(* CoDeSys 2.3 library: InfluxDB_1.0.0.0.lib *)
(* Libraries: BinaryTool_1.0.0.0.lib 25.8.19 15:16:50, TcpIp.lib 31.8.18 23:12:47, STANDARD.LIB 5.6.98 11:03:02, TcBase.lib 14.5.09 11:14:08, TcSystem.lib 7.6.16 10:01:22, TcUtilities.lib 3.2.16 15:08:58 *)

(* Global variable list: Global_Variables *)
VAR_GLOBAL
END_VAR
VAR_GLOBAL CONSTANT
	INFLUX_ROW_LEN : UINT := 350;
	INFLUX_FIFO_SIZE : UINT := 200;
	INFLUX_BUFFER_SIZE : UINT := 1200;
END_VAR

(* Data type *)
TYPE ST_InfluxDB_ConPar :
STRUCT
	sIpv4Address	: STRING	:= '127.0.0.1';
	uPort			: UINT		:= 8086;
	sHostName		: STRING	:= 'localhost';
	sDatabase		: STRING;
	sUser 			: STRING;
	sPassword		: STRING;
END_STRUCT
END_TYPE

(* Data type *)
TYPE ST_InfluxDB_Response :
STRUCT
	sContent		: T_MAXString;
	uCode		: UINT;
	bError		: BOOL;
END_STRUCT
END_TYPE

(* POU F_InfluxDb_BuildHttpPostRequest, ST *)
FUNCTION F_InfluxDb_BuildHttpPostRequest : BOOL
VAR_INPUT
	i_stInfluxDB_ConPar	: ST_InfluxDB_ConPar;
END_VAR
VAR_IN_OUT
	io_sInFluxData	: STRING(INFLUX_FIFO_SIZE);
	io_sBytesToSend	: FB_BinaryTool;
END_VAR
VAR
	nLength             : INT;
END_VAR
F_InfluxDb_BuildHttpPostRequest := F_BinaryTool_WriteString('POST ',io_sBytesToSend);
F_InfluxDb_BuildHttpPostRequest := F_InfluxDB_MakeURL(i_stInfluxDB_ConPar := i_stInfluxDB_ConPar, io_fbBinaryTool := io_sBytesToSend) AND F_InfluxDb_BuildHttpPostRequest;
F_InfluxDb_BuildHttpPostRequest := F_BinaryTool_WriteString(' HTTP/1.1$R$N',io_sBytesToSend) AND F_InfluxDb_BuildHttpPostRequest;
F_InfluxDb_BuildHttpPostRequest := F_BinaryTool_WriteString('Host: ',io_sBytesToSend) AND F_InfluxDb_BuildHttpPostRequest;
F_InfluxDb_BuildHttpPostRequest := F_BinaryTool_WriteString(i_stInfluxDB_ConPar.sHostName,io_sBytesToSend) AND F_InfluxDb_BuildHttpPostRequest;
F_InfluxDb_BuildHttpPostRequest := F_BinaryTool_WriteString(' $R$N',io_sBytesToSend) AND F_InfluxDb_BuildHttpPostRequest;
F_InfluxDb_BuildHttpPostRequest := F_BinaryTool_WriteString('User-Agent: TwinCAT HttpClient$R$N',io_sBytesToSend) AND F_InfluxDb_BuildHttpPostRequest;
F_InfluxDb_BuildHttpPostRequest := F_BinaryTool_WriteString('Content-Type: application/x-www-form-urlencoded$R$N',io_sBytesToSend) AND F_InfluxDb_BuildHttpPostRequest;

(*// Calculate the length of data*)
F_InfluxDb_BuildHttpPostRequest := F_BinaryTool_WriteString('Content-Length: ',io_sBytesToSend) AND F_InfluxDb_BuildHttpPostRequest;
nLength := LEN(io_sInFluxData);
F_InfluxDb_BuildHttpPostRequest := F_BinaryTool_WriteTArg(F_INT(nLength),io_sBytesToSend) AND F_InfluxDb_BuildHttpPostRequest;

(*// Http request headers always end to double new line		*)
F_InfluxDb_BuildHttpPostRequest := F_BinaryTool_WriteString('$R$N$R$N',io_sBytesToSend) AND F_InfluxDb_BuildHttpPostRequest;
(*// Copy the influx data into http request*)
F_InfluxDb_BuildHttpPostRequest := F_BinaryTool_WriteBuffer(ADR(io_sInFluxData),LEN(io_sInFluxData),io_sBytesToSend) AND F_InfluxDb_BuildHttpPostRequest;
(*// Http request body always ends TO new line*)
F_InfluxDb_BuildHttpPostRequest := F_BinaryTool_WriteString('$R$N',io_sBytesToSend) AND F_InfluxDb_BuildHttpPostRequest;


(****** POST Request principle ***********************************************************************

POST /write?db=name HTTP/1.1$R$N
Host: domain.sud $R$N
User-Agent: TwinCAT HttpClient$R$N
Content-Type: application/x-www-form-urlencoded$R$
NContent-Length: 123$R$N$R$N
...Data...$N
$R$N

******************************************************************************************************)
END_FUNCTION

(* POU F_InfluxDB_MakeURL, ST *)
FUNCTION F_InfluxDB_MakeURL : BOOL
VAR_INPUT
	i_stInfluxDB_ConPar	: ST_InfluxDB_ConPar;
END_VAR
VAR_IN_OUT
	io_fbBinaryTool	: FB_BinaryTool;
END_VAR
VAR
END_VAR
F_InfluxDB_MakeURL := F_BinaryTool_WriteString(i_sStringToAppend := '/write?db=', io_fbBinaryTool := io_fbBinaryTool);
F_InfluxDB_MakeURL := F_BinaryTool_WriteString(i_sStringToAppend := i_stInfluxDB_ConPar.sDatabase, io_fbBinaryTool := io_fbBinaryTool) AND F_InfluxDB_MakeURL;

IF i_stInfluxDB_ConPar.sUser <> '' THEN
	F_InfluxDB_makeURL := F_BinaryTool_WriteString(i_sStringToAppend := '&u=', io_fbBinaryTool := io_fbBinaryTool) AND F_InfluxDB_makeURL;
	F_InfluxDB_MakeURL := F_BinaryTool_WriteString(i_sStringToAppend := i_stInfluxDB_ConPar.sUser, io_fbBinaryTool := io_fbBinaryTool) AND F_InfluxDB_MakeURL;
END_IF
IF i_stInfluxDB_ConPar.sPassword <> '' THEN
	F_InfluxDB_makeURL := F_BinaryTool_WriteString(i_sStringToAppend := '&p', io_fbBinaryTool := io_fbBinaryTool) AND F_InfluxDB_makeURL;
	F_InfluxDB_MakeURL := F_BinaryTool_WriteString(i_sStringToAppend := i_stInfluxDB_ConPar.sPassword, io_fbBinaryTool := io_fbBinaryTool) AND F_InfluxDB_MakeURL;
END_IF
END_FUNCTION

(* POU F_InfluxDB_GetTime, ST *)
FUNCTION F_InfluxDB_GetTime : STRING(22)
VAR CONSTANT
	unixTimeFileTimeDiff	: T_ULARGE_INTEGER := (dwHighPart := 16#19DB1DE,dwLowPart := 16#D53E8000);
END_VAR
VAR
	fbGetSystemTime			: GETSYSTEMTIME;
	unixTimeFileTime		: T_ULARGE_INTEGER;
 END_VAR
(****************************************************************************************************************

In TwinCAT we get accure timestamp  via GetSystemTime() FUNCTION block, but it returns so called "filetime"
	filemtime is count of "100 nanoseconds" since 1.1.1601.
	
InfluxDb uses Unix time stamp with accuracy of 1ns. 
	Unix time stamp is seconds since 1.1.1970. 

1.1.1970 - 1.1.1601 in "100 nanoseconds" is 116444736000000000	
	and in Hex 19D B1DE D53E 8000
*******************************************************************************************************************)
fbGetSystemTime( timeLoDW=>unixTimeFileTime.dwLowPart, timeHiDW=>unixTimeFileTime.dwHighPart );  (* "100 nanoseconds" since 1.1.1601. *)
unixTimeFileTime 	:=UInt64Sub64 (unixTimeFileTime,unixTimeFileTimeDiff); (* "100 nanoseconds" since 1.1.1970. *)
F_InfluxDB_GetTime	:= UINT64_TO_STRING (unixTimeFileTime) (* IEC Error when not *);
F_InfluxDB_GetTime 	:= CONCAT(F_InfluxDB_GetTime,'00'); (* *100  and it is nanoseconds since 1.1.1970. *)
END_FUNCTION

(* POU F_InfluxDb_ParseArg, ST *)
FUNCTION F_InfluxDb_ParseArg : BOOL
VAR_INPUT
	i_sNameArg: STRING;
	i_stArg: T_Arg;
	i_sFormatArg: STRING;
END_VAR
VAR_IN_OUT
	io_fbBinaryTool: FB_BinaryTool;
END_VAR
VAR
	udCurrentLen 	: UDINT;
	fbFormatString	: FB_FormatString;
END_VAR
F_InfluxDb_ParseArg := TRUE;
IF i_sNameArg<> '' THEN
	udCurrentLen := F_BinaryTool_Length(io_fbBinaryTool);
	F_InfluxDb_ParseArg := F_BinaryTool_WriteString(',',io_fbBinaryTool);
	F_InfluxDb_ParseArg := F_BinaryTool_WriteString(i_sNameArg,io_fbBinaryTool) AND F_InfluxDb_ParseArg;
	F_InfluxDb_ParseArg := F_BinaryTool_WriteString('=',io_fbBinaryTool) AND F_InfluxDb_ParseArg;
	IF i_sFormatArg <> '' THEN
		fbFormatString(sFormat := i_sFormatArg,arg1:=i_stArg);
		F_InfluxDb_ParseArg := (NOT  fbFormatString.bError) AND F_InfluxDb_ParseArg;
		F_InfluxDb_ParseArg := F_BinaryTool_WriteString(fbFormatString.sOut,io_fbBinaryTool) AND F_InfluxDb_ParseArg;
	ELSE
		F_InfluxDb_ParseArg := F_BinaryTool_WriteTArg(i_stArg,io_fbBinaryTool) AND F_InfluxDb_ParseArg;
	END_IF
END_IF
END_FUNCTION

(* POU F_InfluxDB_ParseHttpResponse, ST *)
FUNCTION F_InfluxDB_ParseHttpResponse : ST_InfluxDB_Response
VAR_IN_OUT
	io_fbBinaryTool: FB_BinaryTool;
END_VAR
VAR
(*
	i				: UDINT;
	headerIndex		: UDINT;
	stHttpResp 		: ST_HTTP_Response;
	pReceivedBytes	: POINTER TO BYTE;
	udNumOfBytes	: UDINT;
	udBytesToCopy	: UDINT;
	start: UDINT;
	arrDummyArray	: ARRAY [0..HTTP_RECEIVE_DATA_ARRAY_SIZE] OF BYTE;
	length: UDINT;
*)
	sLineBreak          	:  STRING :=	'$R$N';
	sDLineBreak          	:  STRING :=	'$R$N$R$N';
	udPos 			:  UDINT;
	udSubPos 		:  INT;
	udOldPos		:  UDINT;
	sHeader 		: T_maxString;
END_VAR
udPos := F_BinaryTool_FindByte(i_pBufferToFind := ADR(sDLineBreak), i_udBufferLen := LEN(sDLineBreak), i_udStartPos := 1, io_fbBinaryTool := io_fbBinaryTool);
F_InfluxDB_ParseHttpResponse.sContent :=F_BinaryTool_ToStringPos(i_udStartPos := udPos+4, i_udEndPos :=F_BinaryTool_Length(io_fbBinaryTool := io_fbBinaryTool), io_fbBinaryTool := io_fbBinaryTool);
F_InfluxDB_ParseHttpResponse.uCode := 0;
F_InfluxDB_ParseHttpResponse.bError := TRUE;

udPos:=1;
udOldPos:=1;
WHILE udPos>0 DO
	udPos := F_BinaryTool_FindByte(i_pBufferToFind := ADR(sLineBreak), i_udBufferLen := LEN(sLineBreak), i_udStartPos := udPos, io_fbBinaryTool := io_fbBinaryTool);
	IF udPos>0 THEN
		sHeader :=F_BinaryTool_ToStringPos(i_udStartPos := udOldPos, i_udEndPos :=udPos-1, io_fbBinaryTool := io_fbBinaryTool);
		udSubPos := FIND (sHeader,'HTTP');
		IF udSubPos > 0 THEN
			sHeader := MID(sHeader,LEN(sHeader),udSubPos+4);
			udSubPos := FIND (sHeader,' ');
			sHeader := MID(sHeader,LEN(sHeader),udSubPos+1);
			udSubPos := FIND (sHeader,' ');
			sHeader := MID(sHeader,udSubPos-1,1);
			F_InfluxDB_ParseHttpResponse.uCode := STRING_TO_UINT (sHeader);
			F_InfluxDB_ParseHttpResponse.bError := F_InfluxDB_ParseHttpResponse.uCode <> 204;
			udPos := 0;
		ELSE
			udPos := udPos+2;
			udOldPos := udPos;
		END_IF
	END_IF;
END_WHILE

(****** POST Response principle A ************************************************************

HTTP/1.1 204 No Content$R$N
Content-Type: application/json$R$N
Request-Id: 2734a929-c5cb-11e9-83ad-0242ac11000d$R$N
X-Influxdb-Build: OSS$R$N
X-Influxdb-Version: 1.7.7$R$N
X-Request-Id: 2734a929-c5cb-11e9-83ad-0242ac11000d$R$N
Date: Fri, 23 Aug 2019 17:26:33 GMT$R$N$R$N

******************************************************************************************************)
(****** POST Response principle B ************************************************************

HTTP/1.1 400 Bad Request$R$N
Content-Type: application/json$R$N
Request-Id: 8f733a77-c5d7-11e9-98aa-0242ac11000d$R$N
X-Influxdb-Build: OSS$R$N
X-Influxdb-Error: unable to parse $'Temperat ursensoren,source=Wohnz immer MW_Real1=123.56,MW_Real2=123.559997558594,MW_Real3=123.559997558594,MW_Real4=123.559997558594,MW_Real5=123.559997558594,MW_Real6=123.559997558594,MW_Real7=123.559997558594,MW_Real8=123.559997558594,MW_Real9=123.559997558594,MW_Real10=123.559997558594 1566586477285000000$': invalid boolean$R$N
X-Influxdb-Version: 1.7.7$R$N
X-Request-Id: 8f733a77-c5d7-11e9-98aa-0242ac11000d$R$N
Date: Fri, 23 Aug 2019 18:55:22 GMT$R$N
Content-Length: 123$R$N$R$N
{"error":"..."}
$N

******************************************************************************************************)
END_FUNCTION

(* POU FB_InfluxDB, ST *)
FUNCTION_BLOCK FB_InfluxDB
VAR_INPUT
END_VAR
VAR_OUTPUT
	o_bBusi					: BOOL := FALSE;
	o_bError				: BOOL := FALSE;
	o_sError				: STRING := '';
END_VAR
VAR_IN_OUT
	io_stInfluxDB_ConPar	: ST_InfluxDB_ConPar;
	io_fbInfluxDB_Fifo 		: FB_InfluxDB_Fifo;
END_VAR
VAR
	fbInfluxDB_Fifo			: FB_InfluxDB_Fifo;
	fbInfluxDB_GetHostname 	: FB_InfluxDB_GetHostname;
	fbSocketConnect			: FB_SocketConnect;
	fbSocketSend			: FB_SocketSend;
	fbSocketReceive			: FB_SocketReceive;
	fbSocketClose			: FB_SocketClose;
	nState					: UINT := 10;
	nRecive					: UINT := 10;
	hSocket					: T_HSOCKET;
	bConnected				: BOOL;

	fbBinaryTool			: FB_BinaryTool;
	sBuffer					: STRING(INFLUX_BUFFER_SIZE) := '';
	stInfluxDB_Response		: ST_InfluxDB_Response;
	io_InfluxDB_ConPar		: BOOL;
END_VAR
fbInfluxDB_GetHostname(i_bStart := FALSE, io_stInfluxDB_ConPar := io_stInfluxDB_ConPar);
fbSocketConnect(bExecute := FALSE, hSocket => hSocket);
fbSocketSend(hSocket := hSocket, bExecute := FALSE);
fbSocketReceive(hSocket := hSocket, bExecute := FALSE);
fbSocketClose(hSocket := hSocket, bExecute := FALSE);

CASE nState OF
10: (* Initial state *)
	IF (io_fbInfluxDB_Fifo.Data) THEN
		io_fbInfluxDB_Fifo.pop();
		o_bBusi				:= TRUE;
		o_bError			:= FALSE;
		o_sError			:= '';
		fbBinaryTool(i_pDestAddr		:= ADR(sBuffer), i_udDestAddrLen	:= SIZEOF(sBuffer), i_udCurrentLen := 0);
		fbInfluxDB_GetHostname(i_bStart := TRUE, io_stInfluxDB_ConPar := io_stInfluxDB_ConPar);
		IF fbInfluxDB_GetHostname.o_bBuisi THEN
			nState 				:= 20;
		ELSIF fbInfluxDB_GetHostname.o_bError THEN
			o_bBusi				:= FALSE;
			o_bError			:= TRUE;
			o_sError			:= CONCAT('Error Get IP: ',UDINT_TO_STRING(fbInfluxDB_GetHostname.o_nErrID));
		ELSE
			IF bConnected THEN
				nState := 50;
			ELSE
				nState := 30;
			END_IF;
		END_IF
	END_IF;

20:
	IF fbInfluxDB_GetHostname.o_bError THEN
		nState 				:= 10;
		o_bBusi				:= FALSE;
		o_bError			:= TRUE;
		o_sError			:= CONCAT('Error Get IP: ',UDINT_TO_STRING(fbInfluxDB_GetHostname.o_nErrID));
	ELSIF NOT fbInfluxDB_GetHostname.o_bBuisi THEN
		IF bConnected THEN
			nState := 50;
		ELSE
			nState := 30;
		END_IF;
	END_IF;

30:	fbSocketConnect(sRemoteHost := io_stInfluxDB_ConPar.sIpv4Address, nRemotePort := io_stInfluxDB_ConPar.uPort,  bExecute := TRUE, tTimeOut := T#10s);
	nState := 40;

40: IF fbSocketConnect.bError THEN
		nState 				:= 10;
		o_bBusi				:= FALSE;
		o_bError			:= TRUE;
		o_sError			:= CONCAT('Error Connect: ',UDINT_TO_STRING(fbSocketConnect.nErrId));
	ELSIF NOT fbSocketConnect.bBusy THEN
		nState 				:= 50;
		bConnected			:= TRUE;
	END_IF;

50:	F_InfluxDb_BuildHttpPostRequest(i_stInfluxDB_ConPar:=io_stInfluxDB_ConPar,io_sInFluxData:=io_fbInfluxDB_Fifo.out,io_sBytesToSend:=fbBinaryTool);
	fbSocketSend(hSocket := hSocket, cbLen := F_BinaryTool_Length(fbBinaryTool) , pSrc := ADR(sBuffer), bExecute := TRUE, tTimeOut := T#10s);
	nState := 60;

60: IF fbSocketSend.bError THEN
		nState 				:= 10;
		bConnected			:= FALSE;
		o_bBusi				:= FALSE;
		o_bError			:= TRUE;
		o_sError			:= CONCAT('Error Connect: ',UDINT_TO_STRING(fbSocketConnect.nErrId));
	ELSIF NOT fbSocketSend.bBusy THEN
		nState 				:= 70;
		fbBinaryTool(i_pDestAddr		:= ADR(sBuffer), i_udDestAddrLen	:= SIZEOF(sBuffer), i_udCurrentLen:=0);
		fbSocketReceive(hSocket := hSocket, cbLen := SIZEOF(sBuffer) , pDest := ADR(sBuffer), bExecute := TRUE, tTimeOut := T#10s);
		nRecive := 10;
	END_IF;

70: IF fbSocketReceive.bError THEN
		nState 				:= 10;
		o_bBusi				:= FALSE;
		o_bError			:= TRUE;
		o_sError			:= CONCAT('Error Connect: ',UDINT_TO_STRING(fbSocketConnect.nErrId));
	ELSIF NOT fbSocketReceive.bBusy THEN
		IF fbSocketReceive.nRecBytes = 0 AND nRecive>0 THEN
			nRecive:= nRecive - 1;
			fbSocketReceive(bExecute := TRUE);
		ELSE
			F_BinaryTool_SetLength(i_udCurrentLen := fbSocketReceive.nRecBytes,io_fbBinaryTool := fbBinaryTool);
			stInfluxDB_Response 	:= F_InfluxDB_ParseHttpResponse(io_fbBinaryTool := fbBinaryTool);
			o_bError				:= stInfluxDB_Response.bError;
			o_sError				:= stInfluxDB_Response.sContent;
			nState 				:= 80;
		END_IF
	END_IF;

80: IF (io_fbInfluxDB_Fifo.Data) THEN
		nState 				:= 10;
	ELSE
		bConnected			:= FALSE;
		fbSocketClose(hSocket := hSocket, bExecute := TRUE, tTimeOut := T#10s);
		nState 				:= 90;
	END_IF;

90: IF fbSocketClose.bError THEN
		nState 				:= 10;
		o_bBusi				:= FALSE;
		o_bError			:= TRUE;
		o_sError			:= CONCAT('Error Connect: ',UDINT_TO_STRING(fbSocketConnect.nErrId));
	ELSIF NOT fbSocketClose.bBusy THEN
		nState 				:= 10;
	END_IF;


END_CASE;
END_FUNCTION_BLOCK

(* POU FB_InfluxDB_Fifo, ST *)
FUNCTION_BLOCK FB_InfluxDB_Fifo
VAR_INPUT
	in					: STRING(INFLUX_ROW_LEN);
END_VAR
VAR_OUTPUT
	Data				: BOOL := FALSE;
	out					: STRING(INFLUX_ROW_LEN);
	error				: BOOL := FALSE;
END_VAR
VAR
	FifoEntries			: ARRAY[1..INFLUX_FIFO_SIZE] OF STRING(INFLUX_ROW_LEN);
	nFirst				: BYTE := 1;
	nLast 				: BYTE := 1;
	nCount				: BYTE := 0;
END_VAR
;
END_FUNCTION_BLOCK
ACTION pop:
IF nCount = 0 THEN
	error := FALSE;
	Data := FALSE;
	RETURN;
END_IF

out := FifoEntries[ nFirst ];
nFirst := SEL( nFirst = INFLUX_FIFO_SIZE, nFirst + 1, 1 );
nCount := nCount - 1;
error := FALSE;
Data := nCount > 0;
END_ACTION
ACTION push:
IF nCount >= INFLUX_FIFO_SIZE THEN
	error := TRUE;
	RETURN;
END_IF

FifoEntries[ nLast ] := in;
nLast := SEL( nLast = INFLUX_FIFO_SIZE, nLast + 1, 1 );

nCount := nCount + 1;
error := FALSE;
Data := TRUE;
END_ACTION

(* POU FB_InfluxDB_GetHostname, ST *)
FUNCTION_BLOCK FB_InfluxDB_GetHostname
VAR_INPUT
	i_bStart : BOOL;
END_VAR
VAR_OUTPUT
	o_bBuisi : BOOL;
	o_bError : BOOL;
	o_nErrID : UDINT;
END_VAR
VAR_IN_OUT
	io_stInfluxDB_ConPar	: ST_InfluxDB_ConPar;
END_VAR
VAR
	fbR_TRIG 				: R_TRIG;
	fbGetHostAddrByName		: FB_GetHostAddrByName;
	nState					: UINT := 10;
END_VAR
CASE nState OF
10: (* Initial state *)
	fbR_TRIG(CLK := i_bStart);
	IF (fbR_TRIG.Q) THEN
			o_bError := FALSE;
			o_bBuisi := TRUE;
			o_nErrID :=	0;
			IF (io_stInfluxDB_ConPar.sHostName = '') THEN
				io_stInfluxDB_ConPar.sHostName := io_stInfluxDB_ConPar.sIpv4Address;
				o_bBuisi := FALSE;
			END_IF
			IF (io_stInfluxDB_ConPar.sIpv4Address='') THEN
				IF io_stInfluxDB_ConPar.sHostName = 'localhost' THEN
					io_stInfluxDB_ConPar.sIpv4Address := '127.0.0.1';
					o_bBuisi := FALSE;
				ELSE
					fbGetHostAddrByName(
						sHostName	:= io_stInfluxDB_ConPar.sHostName,
						tTimeout 	:= T#10S
					);
					nState 		:= 20;
				END_IF;
			ELSE
				o_bBuisi := FALSE;
			END_IF;
	END_IF;
20:
	fbGetHostAddrByName(
		bExecute 	:= FALSE,
	);

	IF fbGetHostAddrByName.bError THEN
		o_bBuisi := FALSE;
		o_bError := TRUE;
		o_nErrId := fbGetHostAddrByName.nErrID;
		nState := 10;
	ELSIF NOT fbGetHostAddrByName.bBusy THEN
		io_stInfluxDB_ConPar.sIpv4Address := fbGetHostAddrByName.sAddr;
		o_bBuisi := FALSE;
		o_bError := FALSE;
		nState := 10;
	END_IF

END_CASE;
END_FUNCTION_BLOCK

(* POU FB_InfluxDB_StoreData, ST *)
FUNCTION_BLOCK FB_InfluxDB_StoreData
VAR_INPUT
	i_sMeasurement: STRING := 'TwinCat';
	i_sSource: STRING := '';
	i_sNameArg1: STRING := '';
	i_stArg1: T_Arg;
	i_sFormatArg1: STRING := '';
	i_sNameArg2: STRING := '';
	i_stArg2: T_Arg;
	i_sFormatArg2: STRING := '';
	i_sNameArg3: STRING := '';
	i_stArg3: T_Arg;
	i_sFormatArg3: STRING := '';
	i_sNameArg4: STRING := '';
	i_stArg4: T_Arg := ();
	i_sFormatArg4: STRING := '';
	i_sNameArg5: STRING := '';
	i_stArg5: T_Arg;
	i_sFormatArg5: STRING := '';
	i_sNameArg6: STRING := '';
	i_stArg6: T_Arg;
	i_sFormatArg6: STRING := '';
	i_sNameArg7: STRING := '';
	i_stArg7: T_Arg;
	i_sFormatArg7: STRING := '';
	i_sNameArg8: STRING := '';
	i_stArg8: T_Arg;
	i_sFormatArg8: STRING := '';
	i_sNameArg9: STRING := '';
	i_stArg9: T_Arg;
	i_sFormatArg9: STRING := '';
	i_sNameArg10: STRING := '';
	i_stArg10: T_Arg;
	i_sFormatArg10: STRING := '';
	i_sTime: STRING := '';
END_VAR
VAR_OUTPUT
	o_bOK: BOOL;
END_VAR
VAR_IN_OUT
	io_fbInfluxDB_Fifo 			: FB_InfluxDB_Fifo;
END_VAR
VAR
	fbBinaryTool: FB_BinaryTool;
	sBuffer: STRING(INFLUX_ROW_LEN);
	udCurrentLen: UDINT;
END_VAR
	fbBinaryTool(i_pDestAddr := ADR(sBuffer), i_udDestAddrLen := SIZEOF(sBuffer), i_udCurrentLen := 0);

	o_bOK := F_BinaryTool_WriteString(i_sMeasurement,fbBinaryTool);

	IF i_sSource <>'' THEN
		o_bOK := F_BinaryTool_WriteString(',source=',fbBinaryTool) AND o_bOK;
		o_bOK := F_BinaryTool_WriteString(i_sSource,fbBinaryTool) AND o_bOK;
	END_IF
	udCurrentLen := F_BinaryTool_Length(fbBinaryTool);
	o_bOK := F_InfluxDb_ParseArg(i_sNameArg := i_sNameArg1,i_stArg := i_stArg1,i_sFormatArg := i_sFormatArg1,io_fbBinaryTool:=fbBinaryTool) AND o_bOK;
	o_bOK := F_InfluxDb_ParseArg(i_sNameArg := i_sNameArg2,i_stArg := i_stArg2,i_sFormatArg := i_sFormatArg2,io_fbBinaryTool:=fbBinaryTool) AND o_bOK;
	o_bOK := F_InfluxDb_ParseArg(i_sNameArg := i_sNameArg3,i_stArg := i_stArg3,i_sFormatArg := i_sFormatArg3,io_fbBinaryTool:=fbBinaryTool) AND o_bOK;
	o_bOK := F_InfluxDb_ParseArg(i_sNameArg := i_sNameArg4,i_stArg := i_stArg4,i_sFormatArg := i_sFormatArg4,io_fbBinaryTool:=fbBinaryTool) AND o_bOK;
	o_bOK := F_InfluxDb_ParseArg(i_sNameArg := i_sNameArg5,i_stArg := i_stArg5,i_sFormatArg := i_sFormatArg5,io_fbBinaryTool:=fbBinaryTool) AND o_bOK;
	o_bOK := F_InfluxDb_ParseArg(i_sNameArg := i_sNameArg6,i_stArg := i_stArg6,i_sFormatArg := i_sFormatArg6,io_fbBinaryTool:=fbBinaryTool) AND o_bOK;
	o_bOK := F_InfluxDb_ParseArg(i_sNameArg := i_sNameArg7,i_stArg := i_stArg7,i_sFormatArg := i_sFormatArg7,io_fbBinaryTool:=fbBinaryTool) AND o_bOK;
	o_bOK := F_InfluxDb_ParseArg(i_sNameArg := i_sNameArg8,i_stArg := i_stArg8,i_sFormatArg := i_sFormatArg8,io_fbBinaryTool:=fbBinaryTool) AND o_bOK;
	o_bOK := F_InfluxDb_ParseArg(i_sNameArg := i_sNameArg9,i_stArg := i_stArg9,i_sFormatArg := i_sFormatArg9,io_fbBinaryTool:=fbBinaryTool) AND o_bOK;
	o_bOK := F_InfluxDb_ParseArg(i_sNameArg := i_sNameArg10,i_stArg := i_stArg10,i_sFormatArg := i_sFormatArg10,io_fbBinaryTool:=fbBinaryTool) AND o_bOK;

	o_bOK := F_BinaryTool_WriteStringPos(' ',udCurrentLen,fbBinaryTool) AND o_bOK;
	o_bOK := F_BinaryTool_WriteString(' ',fbBinaryTool) AND o_bOK;
	IF i_sTime <> '' THEN
		o_bOK := F_BinaryTool_WriteString(i_sTime,fbBinaryTool) AND o_bOK;
	ELSE
		o_bOK := F_BinaryTool_WriteString(F_InfluxDB_GetTime(),fbBinaryTool) AND o_bOK;
	END_IF
	o_bOK := F_BinaryTool_WriteString('$N',fbBinaryTool) AND o_bOK;
	IF (o_bOK) THEN
		io_fbInfluxDB_Fifo.push(in := sBuffer);
	END_IF
END_FUNCTION_BLOCK
